// TIA Portal V20 export
TYPE "UDT_OPC_Analog"
   STRUCT
      Delay : Real;   // Unit:s
      DiffErrorMax : Real;
      DiffErrorMin : Real;
      DiffWarnMax : Real;
      DiffWarnMin : Real;
      Id : Int;
      Offset : Real;
      Gain : Real := 1.0;
      Target : Real;
      Value : Real;
      Update : Bool;
   END_STRUCT;
END_TYPE
